  //================================================================================== 
  // Harmontromics / (C) Copyright (2022) 
  //----------------------------------------------------------------------------------
  // Title:                            按钮点击控制
  // Comment/Function:    根据按下时长，输出不同脉冲信号
  //                     				 按下1s内，输出1个脉冲信号
  //                     				 按下超过1s，已200ms间隔输出脉冲信号
  //                    				 按下超过2s，已100ms间隔输出脉冲信号
  //                    				 按下超过3s，已50ms间隔输出脉冲信号
  //                     			     按下超过5s，已PLC扫描周期间隔输出脉冲信号
  // Library/Family:      (that the source is dedicated to)
  // Author:                 David.Wong
  // Target System: 
  // Engineering:         Sysmac Studio
  // Restrictions:           (OB types, etc.)
  // Requirements:        (hardware, technological package, etc.) 
  //----------------------------------------------------------------------------------
  // Change log table:
  // Version     | Date       | Expert in charge | Changes applied
  //-------------|------------|------------------|------------------------------------
  // 001.000.000 | 2023-8-3  | David.Wong       | First released version
  //            		  |            |                  |              
  //           	  		  |            |                  | 
  //================================================================================== 
IF NOT clickTimer.IN AND CLK THEN
  Q := TRUE;
ELSIF clickTimer.Q THEN //长按超过5s，已PLC扫描周期间隔脉冲输出
  cache := NOT cache;
  Q := cache;
ELSIF clickTimer.ET > T#3s THEN //长按超过3s，已50ms间隔脉冲输出
  Q := timeCache <> TIME_TO_UDINT(clickTimer.ET) / 50;
  timeCache := TIME_TO_UDINT(clickTimer.ET) / 50;
ELSIF clickTimer.ET > T#2s THEN  //长按超过2s，已100ms间隔脉冲输出
  Q := timeCache <> TIME_TO_UDINT(clickTimer.ET) / 100;
  timeCache := TIME_TO_UDINT(clickTimer.ET) / 100;
ELSIF clickTimer.ET > T#1s THEN //长按超过1s，已200ms间隔脉冲输出
  Q := timeCache <> TIME_TO_UDINT(clickTimer.ET) / 200;
  timeCache := TIME_TO_UDINT(clickTimer.ET) / 200;
ELSE
  Q := FALSE;
END_IF;
clickTimer(IN := CLK,
              PT := t#5s);

END_FUNCTION_BLOCK

// ---- Standard/Public/03 HMI/FB_UpdateAxisHmi_RD.TcPOU
FUNCTION_BLOCK FB_UpdateAxisHmi_RD
VAR_IN_OUT
hmi : UDT_AxisHmi_RD; //
vari : ARRAY[*] OF UDT_AxisVar_RD; //
data : ARRAY[*] OF UDT_AxisData_RD; //
number : INT; //编号
END_VAR
VAR
selectPageValueCache : INT; //
index : INT; //
turnPages : FB_TurnPages_RD; //

END_VAR

IF number >0 THEN	
	hmi.display				:= TRUE ;
	IF hmi.number <> number 
		OR selectPageValueCache  <> hmi.selectPageValue[0]
	THEN
		IF hmi.number <> number  THEN
			hmi.selectDisplay:=FALSE;
			hmi.turnPages.value:=0;
		END_IF;
		hmi.number	:= number;
		selectPageValueCache  := hmi.selectPageValue[0];		
		
		hmi.autoVelo			:=	data[number].autoVelo	;
		hmi.manualVelo		:=	data[number].manualVelo	;
		hmi.jogVelo				:=	data[number].jogVelo	;
		hmi.acceleration		:=	data[number].acceleration	;
		hmi.deceleration		:=	data[number].deceleration	;
		hmi.homeDisplay		:=	data[number].homeDisplay	;
		hmi.movehmiNo		:=	vari[number].movehmiNo	;
		FOR index:=1  TO 8 DO			
			IF hmi.selectPageValue[0] + index <= vari[number].movePosNum THEN
				hmi.selectPageValue[index]:=hmi.selectPageValue[0]+index;
				hmi.movePos[index]:= data[number].movePos[ hmi.selectPageValue[0] + index];
			ELSE
				hmi.selectPageValue[index]:=0;
			END_IF;
		END_FOR;	
		hmi.textListNo:=number +1000;
		
	ELSE
		
		data[number].autoVelo			:=	hmi.autoVelo	;
		data[number].manualVelo		:=	hmi.manualVelo	;
		data[number].jogVelo				:=	hmi.jogVelo	;
		data[number].acceleration		:=	hmi.acceleration	;
		data[number].deceleration		:=	hmi.deceleration	;
		data[number].homeDisplay		:=	hmi.homeDisplay	;
		vari[number].powerhmi			:=	hmi.powerhmi	;
		vari[number].halthmi				:=	hmi.halthmi	;
		vari[number].jogForwardhmi	:=	hmi.jogForwardhmi	;
		vari[number].jogBackwardshmi	:=	hmi.jogBackwardshmi	;
		vari[number].homehmi			:=	hmi.homehmi	;
		vari[number].brakehmi			:=	hmi.brakehmi	;
		vari[number].movehmi			:=	hmi.movehmi	;
		hmi.movehmiNo	:= MIN(hmi.movehmiNo	,vari[number].movePosNum);
		vari[number].movehmiNo		:=	hmi.movehmiNo	;
				
		hmi.powerForbidIcon			:=	vari[number].powerForbidIcon	;
		hmi.isPowerOn					:=	vari[number].isPowerOn	;	
		hmi.jogForwardForbidIcon	:=	vari[number].jogForwardForbidIcon	;		
		hmi.jogBackwardsForbidIcon	:=	vari[number].jogBackwardsForbidIcon	;		
		hmi.homeForbidIcon			:=	vari[number].homeForbidIcon	;
		hmi.homeDisplay					:=	vari[number].homeDisplay	;
		hmi.homeDone					:=	vari[number].homeDone	;	
		hmi.brakeForbidIcon			:=	vari[number].brakeForbidIcon	;
		hmi.brake								:=	vari[number].brake	;		
		hmi.moveForbidIcon			:=	vari[number].moveForbidIcon	;
		hmi.brakeState						:=	vari[number].brakeState	;
		hmi.actPos							:=	vari[number].actPos	;
		hmi.actVelo							:=	vari[number].actVelo	;
		hmi.actTorque						:=	vari[number].actTorque	;
		hmi.errorID							:=	vari[number].errorID	;
		hmi.warnID							:=	vari[number].warnID	;		
		hmi.status							:=	vari[number].status	;
		hmi.posUnit							:=	vari[number].posUnit	;
		hmi.veloUnit						:=	vari[number].veloUnit	;
		hmi.accDecUnit					:=	vari[number].accDecUnit	;
		hmi.movePosNum				:=	vari[number].movePosNum	;
		
		FOR index:=0 TO SIZEOF(vari[number].inPos)-1 DO
			hmi.inPosNo := 0;
		    IF 	vari[number].inPos[index] THEN
				hmi.inPosNo := index;
				EXIT;
			END_IF;
		END_FOR;	
		
		FOR index:=1  TO 8 DO
			IF hmi.selectPageValue[0] + index <= vari[number].movePosNum THEN
				data[number].movePos[ hmi.selectPageValue[0] + index] :=hmi.movePos[index];
			END_IF;
		END_FOR;	
		hmi.turnPages.minValue := 0;
     	hmi.turnPages.maxValue := SEL(vari[number].modulo.enable, // 启用模长定位时定位参数显示数量 - 5，定位参数2-6不显示
					                                         vari[number].movePosNum,
					                                         DINT_TO_INT(vari[number].movePosNum - 5));
      	hmi.turnPages.increment := 8;		
		IF hmi.turnPages.prevClick 
			OR hmi.turnPages.nextClick 
			OR  turnPages.value <>  hmi.turnPages.value 
		THEN
			hmi.selectPageValue[0]:= hmi.turnPages.value;
		END_IF;
		turnPages(IN:=hmi.turnPages);
	END_IF;
ELSE
	hmi.display				:= FALSE ;
END_IF;

END_FUNCTION_BLOCK

// ---- Standard/Public/03 HMI/FB_UpdateCycleTimeHmi_RD.TcPOU
FUNCTION_BLOCK FB_UpdateCycleTimeHmi_RD
VAR_IN_OUT
hmi : UDT_Hmi_RD; //
machine : UDT_Machine_RD; //
station : ARRAY[*] OF UDT_Station_RD; //
cycleTime : UDT_CycleTimeHmi_RD; //
number : INT; //编号
END_VAR
VAR
upperBound : INT; //
stationNum : INT; //
index : INT; //
stationIndex : INT; //
fbTurnPages : FB_TurnPages_RD; //
firstRun : BOOL :=TRUE;
END_VAR

  //================================================================================== 
  // Harmontromics / (C) Copyright (2021) 
  //----------------------------------------------------------------------------------
  // Title:               CycleTime
  // Comment/Function:    把各个工站CT和整机CT收集并整理后显示到HMI上，分页显示CT超高显示红色
  // Library/Family:      (that the source is dedicated to)
  // Author:              David.Wong
  // Target System: 
  // Engineering:         TIA Portal (V15.1)
  // Restrictions:        (OB types, etc.)
  // Requirements:        (hardware, technological package, etc.) 
  //----------------------------------------------------------------------------------
  // Change log table:
  // Version     | Date       | Expert in charge | Changes applied
  //-------------|------------|------------------|------------------------------------
  // 001.000.000 | 2021-12-11 | David.Wong       | First released version
  // 001.000.001 | 2022-11-8  | David.Wong       | 增加上下翻页按钮的显示/隐藏
  //             |            |                  |              
  //             |            |                  | 
  //================================================================================== 
SetUp();
CycleTimeHmi();
Visibility();

ACTION CycleTimeHmi:
//--------------------------- CycleTime-------------------------------------------//
  
// 计数之前先清除MAX值
cycleTime.number[0] := machine.machineNo;
cycleTime.cycleTime[0] := machine.cycleTime;
cycleTime.idealCycleTime := TIME_TO_DINT(machine.idealCycleTime);
cycleTime.cycleTimeMin := 0;
cycleTime.cycleTimeMax :=  cycleTime.cycleTime[0];
stationNum := 0;
FOR index := 1 TO upperBound DO
  stationIndex := hmi.includingStationIndex[index];  //获取该工站的索引下标
  // 获取该机器所属工站的CT值，并计数出所有工站最大CT值
  IF stationIndex > 0 THEN
    stationNum := stationNum +1;
    cycleTime.cycleTimeMax := MAX(cycleTime.cycleTimeMax, station[stationIndex].cycleTime);
  END_IF;
END_FOR;
END_ACTION

ACTION SetUp:
//---------------------------SetUp-------------------------------------------//
  IF firstRun THEN
    // 获取数组的上限
    upperBound := SIZEOF(station) -1;   
	firstRun:=FALSE;
  END_IF;
END_ACTION

ACTION Visibility:
//---------------------------- Visibility-------------------------------------------//
// 显示
IF hmi.actPageNo = 110 THEN

	cycleTime.turnPages.minValue:=0;
	cycleTime.turnPages.maxValue:=LINT_TO_INT(MAX(0,stationNum));
	cycleTime.turnPages.increment:=8;
	fbTurnPages(IN:=cycleTime.turnPages);

	FOR index := 1 TO 8 DO
		//显示当前页的工站名称
		cycleTime.number[index] 	:=hmi.includingStationIndex[index + cycleTime.turnPages.value];
		//显示当前页的CT值
		cycleTime.cycleTime[index] :=station[cycleTime.number[index]].cycleTime;
		//当前页的工站CT是否显示
		cycleTime.display[index] 		:=cycleTime.number[index]>0;
	END_FOR;

END_IF;
END_ACTION

END_FUNCTION_BLOCK

// ---- Standard/Public/03 HMI/FB_UpdateInsertHmi_RD.TcPOU
FUNCTION_BLOCK FB_UpdateInsertHmi_RD
VAR_IN_OUT
hmi : UDT_InsertHmi_RD; //
vari : ARRAY[*] OF UDT_InsertVar_RD; //
data : ARRAY[*] OF UDT_InsertData_RD; //
number : INT; //编号
END_VAR
VAR
selectPageValueCache : INT; //
index : INT; //
turnPages : FB_TurnPages_RD; //
activated : Bool; //
posNum : INT; //

END_VAR

IF number >0 THEN	
	posNum:=vari[number].maxCount;
  
	IF hmi.number[0] <> number 
		OR selectPageValueCache  <> hmi.turnPages.value
	THEN
		hmi.number[0]	:= number;
		selectPageValueCache  := hmi.turnPages.value;	
		hmi.selectPinNo:=vari[number].selectPinNo;
		hmi.camSpeed:=data[number].camSpeed;
		FOR index:=1  TO 8 DO			
			IF hmi.turnPages.value + index <= PosNum THEN
				hmi.number [index]:=hmi.turnPages.value + index;
				hmi.enable[index]:= data[number].enable[ hmi.turnPages.value + index];
				hmi.xPosition[index]:= data[number].x.Position[ hmi.turnPages.value + index];
				hmi.yPosition[index]:= data[number].y.Position[ hmi.turnPages.value + index];
				hmi.zPosition[index]:= data[number].z.Position[ hmi.turnPages.value + index];
				hmi.send1Position[index]:= data[number].send1.Position[ hmi.turnPages.value + index];
				hmi.send2Position[index]:= data[number].send2.Position[ hmi.turnPages.value + index];	
				hmi.send3Position[index]:= data[number].send3.Position[ hmi.turnPages.value + index];	
				hmi.send4Position[index]:= data[number].send4.Position[ hmi.turnPages.value + index];	
				hmi.xOffset[index]:= data[number].x.offset[ hmi.turnPages.value + index];
				hmi.yOffset[index]:= data[number].y.offset[ hmi.turnPages.value + index];
				hmi.zOffset[index]:= data[number].z.offset[ hmi.turnPages.value + index];			
				
				hmi.dsplay[index]:=TRUE;
			ELSE
				hmi.number [index]:=0;
				hmi.dsplay[index]:=FALSE;
			END_IF;
			
		END_FOR;		
	ELSE
		IF NOT vari[number].nextPinHmi AND hmi.nextPinHmi THEN
			hmi.selectPinNo:=hmi.selectPinNo +1;
		ELSIF NOT vari[number].previousPinHmi AND hmi.previousPinHmi THEN
			hmi.selectPinNo:=hmi.selectPinNo -1;
		END_IF;
 		IF vari[number].selectPinNo<> hmi.selectPinNo  THEN			
			//vari[number].selectPinNo:=GetSimilarInArray(hmi.selectPinNo,vari[number].pinNo);
			//hmi.selectPinNo:=vari[number].selectPinNo;
			vari[number].selectPinNo:= hmi.selectPinNo;	
		END_IF;
		vari[number].nextPinHmi:=hmi.nextPinHmi;
		vari[number].previousPinHmi:=hmi.previousPinHmi;		
		vari[number].transferMoveHmi:=hmi.transferMoveHmi;		
		vari[number].camNextHmi:=hmi.camNextHmi;		
		vari[number].send1PrevPinHmi:=hmi.send1PrevPinHmi;		
		vari[number].send1NextPinHmi:=hmi.send1NextPinHmi;		
		vari[number].send2PrevPinHmi:=hmi.send2PrevPinHmi;		
		vari[number].send2NextPinHmi:=hmi.send2NextPinHmi;		
		vari[number].send3PrevPinHmi:=hmi.send3PrevPinHmi;		
		vari[number].send3NextPinHmi:=hmi.send3NextPinHmi;				
		vari[number].send4PrevPinHmi:=hmi.send4PrevPinHmi;		
		vari[number].send4NextPinHmi:=hmi.send4NextPinHmi;				
		data[number].camSpeed:=hmi.camSpeed;
		hmi.send1Enable :=vari[number].send1.enable;
		hmi.send2Enable :=vari[number].send2.enable;
		hmi.send3Enable :=vari[number].send3.enable;
		hmi.send4Enable :=vari[number].send4.enable;
		
		hmi.actPinNo :=vari[number].actPinNo;
		hmi.count :=vari[number].count;
		hmi.setCount :=vari[number].setCount;
		hmi.camActPos :=vari[number].cam.actPos;
		hmi.xActPos :=vari[number].x.actPos;
		hmi.yActPos :=vari[number].y.actPos;
		hmi.zActPos :=vari[number].z.actPos;
		hmi.send1ActPos :=vari[number].send1.actPos;
		hmi.send2ActPos :=vari[number].send2.actPos;
		hmi.camSynStatus :=vari[number].cam.synStatus;
		hmi.xSynStatus :=vari[number].x.synStatus;
		hmi.ySynStatus :=vari[number].y.synStatus;
		hmi.zSynStatus :=vari[number].z.synStatus;
		hmi.send1SynStatus :=vari[number].send1.synStatus;
		hmi.send2SynStatus :=vari[number].send2.synStatus;
		FOR index:=1  TO 8 DO
			IF hmi.turnPages.value + index <= PosNum THEN
				IF hmi.send1Position[index] <> 0.0 THEN//送端子1设置值时送端子2\3\4清零
					hmi.send2Position[index]:=0.0;
					hmi.send3Position[index]:=0.0;
					hmi.send4Position[index]:=0.0;
				ELSIF hmi.send2Position[index] <> 0.0 THEN
					hmi.send3Position[index]:=0.0;
					hmi.send4Position[index]:=0.0;
				ELSIF hmi.send3Position[index] <> 0.0 THEN
					hmi.send4Position[index]:=0.0;					
				END_IF;	
				data[number].enable[ hmi.turnPages.value + index]:=hmi.enable[index];
				data[number].x.Position[ hmi.turnPages.value + index]:=hmi.xPosition[index];
				data[number].y.Position[ hmi.turnPages.value + index]:=hmi.yPosition[index];
				data[number].z.Position[ hmi.turnPages.value + index]:=hmi.zPosition[index];
				data[number].send1.Position[ hmi.turnPages.value + index]:=hmi.send1Position[index];
				data[number].send2.Position[ hmi.turnPages.value + index]:=hmi.send2Position[index];
				data[number].send3.Position[ hmi.turnPages.value + index]:=hmi.send3Position[index];
				data[number].send4.Position[ hmi.turnPages.value + index]:=hmi.send4Position[index];
				data[number].x.offset[ hmi.turnPages.value + index]:=hmi.xOffset[index];
				data[number].y.offset[ hmi.turnPages.value + index]:=hmi.yOffset[index];
				data[number].z.offset[ hmi.turnPages.value + index]:=hmi.zOffset[index];
			
				hmi.dsplay[index]:=TRUE;
			ELSE
				hmi.number [index]:=0;
				hmi.dsplay[index]:=FALSE;
			END_IF;
		END_FOR;	
		hmi.turnPages.minValue := 0;
     	hmi.turnPages.maxValue :=	posNum -1;
      	hmi.turnPages.increment := 8;		
		turnPages(IN:=hmi.turnPages);

	END_IF;
ELSE
	hmi.number[0]:=0;
END_IF;

END_FUNCTION_BLOCK

// ---- Standard/Public/03 HMI/FB_UpdateProduceHmi_RD.TcPOU
FUNCTION_BLOCK FB_UpdateProduceHmi_RD
VAR_IN_OUT
hmi : UDT_ProduceHmi_RD; //
machine : ARRAY[*] OF UDT_Machine_RD; //
vari : ARRAY[*] OF UDT_ProduceVar_RD; //
data : ARRAY[*] OF UDT_ProduceData_RD; //
badVar : ARRAY[*] OF UDT_BadVar_RD; //
badData : ARRAY[*] OF UDT_BadData_RD; //
number : INT; //编号
END_VAR

VAR
numberCache : INT; //
goodExecuteCache : Array[0..99] of Bool; //
activated : Bool; //
badExecuteCache : Array[0..99] of Bool; //
badProducts : Array[0..99] of DInt; //
badList : Array[0..99] of Int; //
badSortList : Array[0..99] of Int; //
refresh : Bool; //
pageNo : Int; //
badTypeNum : Int; //
setUpTimer : TON; //
sortModeCache : Int; //
percentModeCache : Int; //
setUpCache : Bool; //
turnPages : FB_TurnPages_RD; //
index : DInt; //
index1 : DInt; //
index2 : DInt; //
temp : DInt; //
No : Int; //
fbTurnPages : FB_TurnPages_RD; //
END_VAR

VAR CONSTANT
MAX_CONTINUOUS  : INT := 99;//最大连续不良报警数量
MAX_CUMULATIVE  : INT := 10;//最大累计不良报警数量n
MAX_CUMULATIVE_RANGE : INT := 999;//最大累计不良计算范围m
END_VAR

IF number >0 THEN
	IF numberCache <> number THEN
		numberCache := number;
				
		hmi.sortMode						:=vari[number].sortMode;
		hmi.percentMode				:=vari[number].percentMode;
	ELSE
		
		badList								:=vari[number].badList;
		badTypeNum					:=vari[number].badTypeNum;
		vari[number].allClearHmi				:=hmi.allClearHmi;
		vari[number].sortMode				:=hmi.sortMode;
		vari[number].percentMode			:=hmi.percentMode;

		IF  hmi.sortMode < 0 OR hmi.sortMode > 2 THEN
			hmi.sortMode :=0;
		END_IF;
		
		// 超过30s自动退出设定模式
		setUpTimer(IN := hmi.setUp,
							PT := t#30S);
		IF setUpTimer.Q THEN
			hmi.setUp := FALSE;
		END_IF;
  
		 //不良显示
		 // 当前不良分类数量多少
		FOR index := 1 TO badTypeNum DO
			No := badList[index];
			badProducts[No] := badData[No].quantity;
		END_FOR;
		
		//不良排序方式
        CASE hmi.sortMode OF
          1:  //根据不良率从大到小排序
            FOR index := 1 TO badTypeNum DO
              temp := badProducts[1];
              badSortList[index] := 1;
              FOR index1 := 1 TO badTypeNum - 1 DO
                IF badProducts[badList[index1 + 1]] > temp THEN
                  temp := badProducts[badList[index1 + 1]];
                  badSortList[index] := badList[index1 + 1];
                END_IF;
                IF index1 = badTypeNum - 1 THEN
                  badProducts[badSortList[index]] := -1;
                END_IF;
              END_FOR;
            END_FOR;
            
          2: //根据不良率从小到大排序
            FOR index := 1 TO badTypeNum DO
              temp := badProducts[1];
              badSortList[index] := 1;
              FOR index1 := 1 TO badTypeNum - 1 DO
                IF badProducts[badList[index1 + 1]] < temp THEN
                  temp := badProducts[badList[index1 + 1]];
                  badSortList[index] := badList[index1 + 1];
                END_IF;
                IF index1 = badTypeNum - 1 THEN
                  badProducts[badSortList[index]] := 99999;
                END_IF;
              END_FOR;
            END_FOR;
          ELSE  //默认排序根据不良类型序号
            FOR index := 1 TO badTypeNum DO
              badSortList[index] := badList[index];
            END_FOR;
        END_CASE;
		

		
        //滚动条控制
		hmi.turnPages.minValue:=0;
		hmi.turnPages.maxValue:=badTypeNum;
		hmi.turnPages.increment:=5;
		fbTurnPages(IN:=hmi.turnPages,
							value=>pageNo);
		FOR index :=1 TO 5 DO
			hmi.badShow[index].display:=badList[index + pageNo] > 0;
		END_FOR;
		
        //进入报警设置中
		badTypeNum:=vari[number].badTypeNum;
        IF hmi.setUp THEN
			FOR index :=1 TO 5 DO
				hmi.badShow[index].setUpDisplay:=badList[index + pageNo] > 0;
			END_FOR;
			FOR index := 1 TO MIN(badTypeNum,5) DO   //显示当前5个，小于5个显示实际数量
				No := badSortList[index + pageNo];
				IF NOT setUpCache AND hmi.setUp
					OR fbTurnPages.change
					OR sortModeCache <> hmi.sortMode
				THEN  //进入设置中上升沿或翻页后执行一次 Data->Show	
            		hmi.badShow[index].number := badSortList[index + pageNo];
					hmi.badShow[index].continuous := badData[No].continuous;
					hmi.badShow[index].cumulative := badData[No].cumulative;
					hmi.badShow[index].cumulativeRange := badData[No].cumulativeRange;
				ELSE//其它时候HMI修改值写入Data Show->Data
					hmi.badShow[index].continuous := LIMIT(hmi.badShow[index].continuous,0, MAX_CONTINUOUS);
					hmi.badShow[index].cumulativeRange := LIMIT(hmi.badShow[index].cumulativeRange,0,MAX_CUMULATIVE_RANGE);
					hmi.badShow[index].cumulative := LIMIT(hmi.badShow[index].cumulative,0,LINT_TO_INT( MIN(MAX_CUMULATIVE,hmi.badShow[index].cumulativeRange)));
					badData[No].continuous := hmi.badShow[index].continuous;
					badData[No].cumulative := hmi.badShow[index].cumulative;
					badData[No].cumulativeRange := hmi.badShow[index].cumulativeRange;
				END_IF;
			END_FOR;
        ELSE//不在报警设置中
			FOR index :=1 TO 5 DO
				hmi.badShow[index].setUpDisplay:=FALSE;
			END_FOR;
          FOR index := 1 TO MIN(badTypeNum,5) DO //显示当前5个，小于5个显示实际数量
            No := badSortList[index + pageNo];
            hmi.badShow[index].number := No;
            hmi.badShow[index].quantity := badData[No].quantity;
            hmi.badShow[index].rate := badVar[No].badRatio;
          END_FOR;
          
		  	hmi.badMax	 		:= vari[number].badMax;
			hmi.badMin 		:= 0;
			setUpCache 		:= hmi.setUp;
			hmi.goodValue 	:=  data[number].goodValue;
			hmi.badValue 		:=  data[number].badValue;
			hmi.totalValue	 	:=  data[number].totalValue;
			hmi.cumulativeValue 		:=  data[number].cumulativeValue;

			hmi.yieldRatio  	:=data[number].yieldRatio;
			hmi.badRatio 		:=data[number].badRatio;
			hmi.pieChart[1]	:= data[number].yieldRatio;
			hmi.pieChart[0]	:= data[number].badRatio;
		  
		  
		  
        END_IF;	
		setUpCache := hmi.setUp;
		sortModeCache	:= hmi.sortMode;


	END_IF;
	
	//连续不良报警
	FOR index2:=0 TO SIZEOF(badVar) BY 1 DO
		hmi.continuousAlarm[index2]:=badVar[index2].continuousAlarm;
		hmi.cumulativeAlarm[index2]:=badVar[index2].cumulativeAlarm;
	END_FOR;
	
END_IF;

END_FUNCTION_BLOCK

// ---- Standard/Unit/06 Axis/FB_NCI.TcPOU
FUNCTION_BLOCK FB_NCI
VAR_INPUT
END_VAR
VAR_OUTPUT
END_VAR
VAR
END_VAR

END_FUNCTION_BLOCK
